PROGRAM MAIN
VAR
END_VAR

END_PROGRAM

(* stored: Version 1.1.0.1
   POU MAIN: Id {0093ae30-d958-4f17-bd94-15a628051bf7} *)
